FUNCTION_BLOCK GENERAL_DATA_SENDER (* Send data that all machine axel will use *)
  (* Standard: 61499-2 *)
  (* Version 1.0, 17-04-2012, GASR, Universidade do Estado de Santa Catarina *)
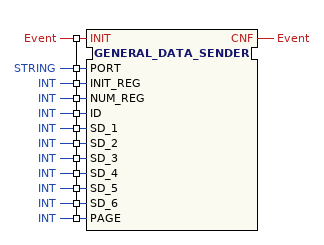
  EVENT_INPUT
    INIT WITH PORT, INIT_REG, NUM_REG, ID, SD_1, SD_2, SD_3, SD_4, SD_5, SD_6, PAGE; (* Initialize service *)
  END_EVENT
  EVENT_OUTPUT
    CNF; (* Execution confirmed *)
  END_EVENT
  VAR_INPUT
    PORT : STRING; (* Ethernet local port *)
    INIT_REG : INT; (* Initial register *)
    NUM_REG : INT; (* Number of registers *)
    ID : INT; (* Process id *)
    SD_1 : INT; (* Parameter 1 *)
    SD_2 : INT; (* Parameter 2 *)
    SD_3 : INT; (* Parameter 3 *)
    SD_4 : INT; (* Parameter 4 *)
    SD_5 : INT; (* Parameter 5 *)
    SD_6 : INT; (* Parameter 6 *)
    PAGE : INT; (* Change "page" parameter *)
  END_VAR
  SERVICE GENERAL_DATA_SENDER/MACHINE (* Data publication service *)
    SEQUENCE normal_data_transfer
      GENERAL_DATA_SENDER.INIT(PORT,INIT_REG,NUM_REG,ID,SD_1,SD_2,SD_3,SD_4,SD_5,SD_6,SD_7,SD_8,SD_9,SD_10,PAGE) -> MACHINE.();
    END_SEQUENCE
  END_SERVICE
END_FUNCTION_BLOCK
